// TIA Portal V20 export
FUNCTION_BLOCK "FB_LoaderShuttle2"   // FB205, SCL
{ S7_Optimized_Access := 'TRUE' }
// stored: AutoNumber false, MemoryReserve 100, SetENOAutomatically false
   VAR_INPUT
      iGripperReserved : Bool;
      iGripperReleased : Bool;
      iShuttleMoving : Bool;
      iShuttleInPos : Bool;
      iAxisV_Moving : Bool;
      iAxisV_InPos : Bool;
      iAxisW_Moving : Bool;
      iAxisW_InPos : Bool;
   END_VAR
   VAR_OUTPUT
      oExtGateOpenReq : Bool;
      oExtGateCloseReq : Bool;
      oIntGateOpenReq : Bool;
      oIntGateCloseReq : Bool;
      oLoadGripperCloseReq : Bool;
      oUnloadGripperOpenReq : Bool;
      oBlowingReq : Bool;
      oShuttleStartReq : Bool;
      oShuttlePosSetPoint : Real;
      oAxisVStartReq : Bool;
      oAxisVPosSetPoint : Real;
      oAxisWStartReq : Bool;
      oAxisWPosSetPoint : Real;
   END_VAR
   VAR
      sMain : "FB_Main";
      sShuttleInt { S7_SetPoint := 'True'} : "FB_ShuttleInt";
      sShuttleExt { S7_SetPoint := 'True'} : "FB_ShuttleExt";
      sControlIn { S7_SetPoint := 'True'} : "FB_PartControl";
      sControlOut { S7_SetPoint := 'True'} : "FB_PartControl";
      sBlowing { S7_SetPoint := 'True'} : "FB_Blowing";
      sIntLoadUnload { S7_SetPoint := 'True'} : "FB_IntLoadUnload";
      sExtLoadUnload { S7_SetPoint := 'True'} : "FB_ExtLoadUnload";
      sBwLoadUnload { S7_SetPoint := 'True'} : "FB_BwLoadUnload";
      sBwControlIn { S7_SetPoint := 'True'} : "FB_BwControl";
      sActPartControlIn { S7_SetPoint := 'True'} : "FB_ActControl";
      sActPartControlout { S7_SetPoint := 'True'} : "FB_ActControl";
      sActBwControlIn { S7_SetPoint := 'True'} : "FB_ActControl";
      sIntLoadUnloadOP { S7_SetPoint := 'True'} : "FB_IntLoadUnloadOP";
      sBwConsecutiveCtrl_1 { S7_SetPoint := 'True'} : "FB_Consecutive";
      sBwConsecutiveCtrl { S7_SetPoint := 'True'} : "FB_Consecutive";
      sShuttlePosInt { S7_SetPoint := 'True'} : Bool;
      sShuttlePosSas : Bool;
      sShuttlePosExt : Bool;
      sGripper_OK : Bool;
      sExtLoaderInSafePos : Bool;
      sIntLoaderInSafePos : Bool;
      sBwLoaderInSafePos : Bool;
      sRT_PartControlInMissing : R_TRIG;
      sRT_PartControlInExtra : R_TRIG;
      sRT_PartControlOutMissing : R_TRIG;
      sRT_PartControlOutExtra : R_TRIG;
      sRT_BwControlInMissing : R_TRIG;
      sRT_BwControlInExtra : R_TRIG;
      sStepPauseSeq { S7_SetPoint := 'True'} : Bool;
   END_VAR
   VAR_TEMP
      tAxis_U_Position : Struct
         ExtLoadUnloadAuto : Bool;
         ExtLoadUnloadManu : Bool;
         PartControl : Bool;
         BwLoad : Bool;
         BwUnload : Bool;
         BwControl : Bool;
         IntLoadUnload : Bool;
         Blowing : Bool;
         IntLoadUnloadOP : Bool;
      END_STRUCT;
      tAxis_V_Position : Struct
         LoadUnload : Bool;
         Safe : Bool;
         Blowing : Bool;
      END_STRUCT;
      tAxis_W_Position : Struct
         LoadUnload : Bool;
         Safe : Bool;
         Approach : Bool;
         Blowing : Bool;
      END_STRUCT;
   END_VAR
BEGIN
   REGION Shuttle 2 position
       // Init Position
       #sShuttlePosInt := FALSE;
       #sShuttlePosSas := FALSE;
       #sShuttlePosExt := FALSE;

       // Check Shuttle (U2 Axis) position
       IF "DB_AxisPosition".sAxis06_U2."$AA_IM" < "DB_AxisPosMachinePLC".Axis_U2.IntGateExt THEN
           #sShuttlePosExt := TRUE;
       ELSIF "DB_AxisPosition".sAxis06_U2."$AA_IM" > "DB_AxisPosMachinePLC".Axis_U2.ExtGateInt THEN
           #sShuttlePosInt := TRUE;
       ELSE
           #sShuttlePosSas := TRUE;
       END_IF;
   END_REGION

   REGION Position Check
       REGION Axis U2
           // Position : External Load / Unload Auto
           "FC_PositionCheck"(iAxisCurrentPos := "DB_AxisPosition".sAxis06_U2."$AA_IM",
                              iAxisTargetPos := "DB_AxisPosMachinePLC".Axis_U2.ExtLoadUnloadAuto,
                              iTolMin := 0.001,
                              iTolMax := 0.001,
                              iInPos => #tAxis_U_Position.ExtLoadUnloadAuto);

           // Position : External Load / Unload Manu
           "FC_PositionCheck"(iAxisCurrentPos := "DB_AxisPosition".sAxis06_U2."$AA_IM",
                              iAxisTargetPos := "DB_AxisPosMachinePLC".Axis_U2.ExtLoadUnloadManu,
                              iTolMin := 0.001,
                              iTolMax := 0.001,
                              iInPos => #tAxis_U_Position.ExtLoadUnloadManu);

           // Position : Part Control
           "FC_PositionCheck"(iAxisCurrentPos := "DB_AxisPosition".sAxis06_U2."$AA_IM",
                              iAxisTargetPos := "DB_AxisPosMachinePLC".Axis_U2.PartControl,
                              iTolMin := 0.001,
                              iTolMax := 0.001,
                              iInPos => #tAxis_U_Position.PartControl);

           // Position : Backwall Load
           "FC_PositionCheck"(iAxisCurrentPos := "DB_AxisPosition".sAxis06_U2."$AA_IM",
                              iAxisTargetPos := "DB_AxisPosMachinePLC".Axis_U2.BwLoad,
                              iTolMin := 0.001,
                              iTolMax := 0.001,
                              iInPos => #tAxis_U_Position.BwLoad);

           // Position : Backwall Unload
           "FC_PositionCheck"(iAxisCurrentPos := "DB_AxisPosition".sAxis06_U2."$AA_IM",
                              iAxisTargetPos := "DB_AxisPosMachinePLC".Axis_U2.BwUnLoad,
                              iTolMin := 0.001,
                              iTolMax := 0.001,
                              iInPos => #tAxis_U_Position.BwUnload);

           // Position : Backwall Control
           "FC_PositionCheck"(iAxisCurrentPos := "DB_AxisPosition".sAxis06_U2."$AA_IM",
                              iAxisTargetPos := "DB_AxisPosMachinePLC".Axis_U2.BwControl,
                              iTolMin := 0.001,
                              iTolMax := 0.001,
                              iInPos => #tAxis_U_Position.BwControl);

           // Position : Internal Load / Unload
           "FC_PositionCheck"(iAxisCurrentPos := "DB_AxisPosition".sAxis06_U2."$AA_IM",
                              iAxisTargetPos := "DB_AxisPosMachinePLC".Axis_U2.IntLoadUnload,
                              iTolMin := 0.001,
                              iTolMax := 0.001,
                              iInPos => #tAxis_U_Position.IntLoadUnload);

           // Position : Internal Load / Unload OP
           "FC_PositionCheck"(iAxisCurrentPos := "DB_AxisPosition".sAxis06_U2."$AA_IM",
                              iAxisTargetPos := "DB_AxisPosMachinePLC".Axis_U2.IntLoadUnloadOP,
                              iTolMin := 0.001,
                              iTolMax := 0.001,
                              iInPos => #tAxis_U_Position.IntLoadUnloadOP);

           // Position : Blowing (Undrilled part)
           "FC_PositionCheck"(iAxisCurrentPos := "DB_AxisPosition".sAxis06_U2."$AA_IM",
                              iAxisTargetPos := "DB_AxisPosMachinePLC".Axis_U2.Blowing,
                              iTolMin := 0.001,
                              iTolMax := 0.001,
                              iInPos => #tAxis_U_Position.Blowing);
       END_REGION

       REGION Axis V
           // Position : Load / Unload Auto
           "FC_PositionCheck"(iAxisCurrentPos := "DB_AxisPosition".sAxis07_V."$AA_IM",
                              iAxisTargetPos := "DB_AxisPosMachinePLC".Axis_V.Shuttle_2.LoadUnload,
                              iTolMin := 0.001,
                              iTolMax := 0.001,
                              iInPos => #tAxis_V_Position.LoadUnload);

           // Position : Safe
           "FC_PositionCheck"(iAxisCurrentPos := "DB_AxisPosition".sAxis07_V."$AA_IM",
                              iAxisTargetPos := "DB_AxisPosMachinePLC".Axis_V.Safe,
                              iTolMin := 0.001,
                              iTolMax := 0.001,
                              iInPos => #tAxis_V_Position.Safe);

           // Position : Blowing
           "FC_PositionCheck"(iAxisCurrentPos := "DB_AxisPosition".sAxis07_V."$AA_IM",
                              iAxisTargetPos := "DB_AxisPosMachinePLC".Axis_V.Shuttle_2.Blowing,
                              iTolMin := 0.001,
                              iTolMax := 0.001,
                              iInPos => #tAxis_V_Position.Blowing);
       END_REGION

       REGION Axis W
           // Position : Load / Unload Auto
           "FC_PositionCheck"(iAxisCurrentPos := "DB_AxisPosition".sAxis08_W."$AA_IM",
                              iAxisTargetPos := "DB_AxisPosMachinePLC".Axis_W.Shuttle_2.LoadUnload,
                              iTolMin := 0.001,
                              iTolMax := 0.001,
                              iInPos => #tAxis_W_Position.LoadUnload);

           // Position : Safe
           "FC_PositionCheck"(iAxisCurrentPos := "DB_AxisPosition".sAxis08_W."$AA_IM",
                              iAxisTargetPos := "DB_AxisPosMachinePLC".Axis_W.Safe,
                              iTolMin := 0.001,
                              iTolMax := 0.001,
                              iInPos => #tAxis_W_Position.Safe);

           // Position : Approach (confondu avec load/unload)
           "FC_PositionCheck"(iAxisCurrentPos := "DB_AxisPosition".sAxis08_W."$AA_IM",
                              iAxisTargetPos := "DB_AxisPosMachinePLC".Axis_W.Shuttle_2.Approach,
                              iTolMin := 0.001,
                              iTolMax := 0.001,
                              iInPos => #tAxis_W_Position.Approach);

           // Position : Blowing
           "FC_PositionCheck"(iAxisCurrentPos := "DB_AxisPosition".sAxis08_W."$AA_IM",
                              iAxisTargetPos := "DB_AxisPosMachinePLC".Axis_W.Shuttle_2.Blowing,
                              iTolMin := 0.001,
                              iTolMax := 0.001,
                              iInPos => #tAxis_W_Position.Blowing);
       END_REGION
   END_REGION

   REGION Step Pause Sequence
       #sStepPauseSeq := "LBP_ModeGroup".E_JOG
       OR "DB_CycleStartStop".sResquestStopNextCycle
       OR "LBP_Chan1".E_M01;

       #sMain.iStepPause := #sStepPauseSeq;
       #sShuttleInt.iStepPause := #sStepPauseSeq;
       #sShuttleExt.iStepPause := #sStepPauseSeq;
       #sIntLoadUnload.iStepPause := #sStepPauseSeq;
       #sIntLoadUnloadOP.iStepPause := #sStepPauseSeq;
       #sControlIn.iStepPause := #sStepPauseSeq;
       #sControlOut.iStepPause := #sStepPauseSeq;
       #sBwLoadUnload.iStepPause := #sStepPauseSeq;
       #sBwControlIn.iStepPause := #sStepPauseSeq;
       #sBlowing.iStepPause := #sStepPauseSeq;
       #sActPartControlIn.iStepPause := FALSE;
       #sActPartControlout.iStepPause := FALSE;
       #sActBwControlIn.iStepPause := FALSE;
   END_REGION

   REGION Main
       // Gripper prêt à Charger / Décharger une pièce
       #sGripper_OK :=
       ((("DB_PartManagement".sPosition.sShuttle2.Undrilled.Presence.Part AND NOT "DB_PartManagement".sPosition.sGripper.Undrilled.Presence.Part AND "DB_GestionGripper".sUndrilledGripper.oStateOpen) OR NOT "DB_PartManagement".sPosition.sShuttle2.Undrilled.Presence.Part)
       AND (("DB_PartManagement".sPosition.sGripper.Drilled.Presence.Part AND NOT "DB_PartManagement".sPosition.sShuttle2.Drilled.Presence.Part) OR NOT "DB_PartManagement".sPosition.sGripper.Drilled.Presence.Part));

       // Loader INT in Safe Position
       #sIntLoaderInSafePos := "DB_AxisPosition".sAxis07_V."$AA_IM" >= "DB_AxisPosMachinePLC".Axis_V.Safe
       OR ("DB_AxisPosition".sAxis07_V."$AA_IM" < "DB_AxisPosMachinePLC".Axis_V.Safe AND "DB_AxisPosition".sAxis08_W."$AA_IM" >= "DB_AxisPosMachinePLC".Axis_W.Safe);

       // Loader EXT in Safe Position
       #sExtLoaderInSafePos := "DB_SonplasMain".sSonplasLoader.iOperateInOutCollision;

       // BW Loader in Safe Position
       #sBwLoaderInSafePos := "DB_BwLoaderExchange".Inputs.BwLoaderInSafePos;

       // Test Stop after Emptying with only one Shuttle
       IF ("DB_WorkingModes".sEmptying
           AND NOT "DB_LoaderShuttle1".sMain.iJobReq
           AND "DB_PartManagement".sPosition.sPartNumber.Total <= 1) THEN
           #sMain.iJobReq := FALSE;
       END_IF;
       // Test Stop after Emptying with two Shuttle
       IF ("DB_WorkingModes".sEmptying
           AND "DB_LoaderShuttle1".sMain.iJobReq
           AND #sMain.sCurrent_Step_NB = 122
           AND "DB_PartManagement".sPosition.sPartNumber.Total <= 2) THEN
           #sMain.iJobReq := FALSE;
       END_IF;

       #sMain(iStartSeqCond := "DB_PowerOn".sMachineReadySoft AND NOT "MCP1_In".reset,
              iJobReq := #sMain.iJobReq,      
              iShuttleINT := #sShuttlePosInt,
              iShuttleSAS:= #sShuttlePosSas,
              iShuttleEXT := #sShuttlePosExt,
              iGripperReserved := #iGripperReserved,
              iGripperReleased := #iGripperReleased,
              iShuttleUndrilledPart:= "DB_PartManagement".sPosition.sShuttle2.Undrilled.Presence.Part,
              iShuttleDrilledPart:= "DB_PartManagement".sPosition.sShuttle2.Drilled.Presence.Part,
              iShuttleUndrilledBw:= "DB_PartManagement".sPosition.sShuttle2.Undrilled.Presence.BW,
              iShuttleDrilledBw:= "DB_PartManagement".sPosition.sShuttle2.Drilled.Presence.BW,
              iPartCtrlInOK:=#sControlIn.oPartControlOK,
              iPartCtrlInNOK:=#sControlIn.oPartControlNOK,
              iPartCtrlInContinuationStep:=#sActPartControlIn.oContinuationStep,
              iPartCtrlInRestartStep:=#sActPartControlIn.oRestartStep,
              iPartCtrlOutOK:=#sControlOut.oPartControlOK,
              iPartCtrlOutNOK:=#sControlOut.oPartControlNOK,
              iPartCtrlOutContinuationStep:=#sActPartControlout.oContinuationStep,
              iPartCtrlOutRestartStep:=#sActPartControlout.oRestartStep,
              iBwCtrlInOK:=#sBwControlIn.oBwControlOK,
              iBwCtrlInNOK:=#sBwControlIn.oBwControlNOK,
              iBwCtrlInContinuationStep:=#sActBwControlIn.oContinuationStep,
              iBwCtrlInRestartStep:=#sActBwControlIn.oRestartStep,
              iGripperOK:=#sGripper_OK,
              iNC_NoNeedAxis:=NOT "DB_CommPLC_ISO".sAxisManagedByNC,
              iExtLoaderInSafePos:=#sExtLoaderInSafePos,
              iIntLoaderInSafePos:=#sIntLoaderInSafePos,
              iBwLoaderInSafePos:=#sBwLoaderInSafePos,
              iOnePieceMode:="DB_WorkingModes".sOnePiece,
              iPLC_DateAndTime := "DB_ReadDateAndTime".sDateAndTime,
              iStepPause:=#sMain.iStepPause,
              oGripperAxisRequest => #sMain.oGripperAxisRequest,
              oGripperAxisRelease => #sMain.oGripperAxisRelease,
              oNoExtLoad=>#sMain.oNoExtLoad,
              oBwLoadReq=> #sMain.oBwLoadReq,
              oBwUnloadReq=> #sMain.oBwUnloadReq,
              ioShuttleIntSeq := #sShuttleInt.sInterface,
              ioShuttleExtSeq := #sShuttleExt.sInterface,
              ioControlInSeq := #sControlIn.sInterface,
              ioControlOutSeq := #sControlOut.sInterface,
              ioBlowingSeq:=#sBlowing.sInterface,
              ioIntLoadUnloadSeq := #sIntLoadUnload.sInterface,
              ioIntLoadUnloadOP_Seq:=#sIntLoadUnloadOP.sInterface,
              ioExtLoadUnloadSeq := #sExtLoadUnload.sInterface,
              ioBWLoadUnloadSeq := #sBwLoadUnload.sInterface,
              ioBWControlSeq := #sBwControlIn.sInterface,
              ioActPartControlInSeq:= #sActPartControlIn.sInterface,
              ioActPartControlOutSeq:= #sActPartControlout.sInterface,
              ioActBwControlInSeq:= #sActBwControlIn.sInterface);
   END_REGION

   REGION Msg Sequence Fault
       // Msg 700015 Shuttle 2 Sequence Fault
       IF #sMain.sCurrent_Step_NB = 999 THEN
           "LBP_AlarmMsgs".UserA[00].A70UUxx[15] := TRUE;
       END_IF;
   END_REGION

   REGION Shuttle 2 INT
       // Position INT :
       //  If Blowing : Pos. Blowing else Pos. Load/Unload
       IF "DB_LoaderOptions".Blowing.Disabled THEN
           #sShuttleInt.iShuttlePosIntSetPoint := "DB_AxisPosMachinePLC".Axis_U2.IntLoadUnload;
       ELSE
           #sShuttleInt.iShuttlePosIntSetPoint := "DB_AxisPosMachinePLC".Axis_U2.Blowing;
       END_IF;

       #sShuttleInt(iStartSeqCond := (#sMain.iStartSeqCond AND NOT #sShuttleInt.sInterface.Error AND NOT "DB_LoaderShuttle1".sShuttleInt.sInterface.SequenceRun AND #sShuttleInt.sInterface.StartRequest),
                    iJobReq := #sShuttleInt.sInterface.StartRequest,
                    iIntGateOpened := "DB_DigitalInputs".sInternalGateOpened.sSWStatus,
                    iIntGateClosed := "DB_DigitalInputs".sInternalGateLocked.sSWStatus,
                    iExtGateOpened := "DB_DigitalInputs".sExternalGateOpened.sSWStatus,
                    iExtGateClosed := "DB_DigitalInputs".sExternalGateLocked.sSWStatus,
                    iShuttlePosInt := #sShuttlePosInt,
                    iShuttlePosSas := #sShuttlePosSas,
                    iShuttlePosExt := #sShuttlePosExt,
                    iShuttlePosIntSetPoint := #sShuttleInt.iShuttlePosIntSetPoint,
                    iShuttlePosSasSetPoint := "DB_AxisPosMachinePLC".Axis_U2.Sas,
                    iShuttleMoving := #iShuttleMoving,
                    iShuttleInPos := #iShuttleInPos,
                    iIntLoaderInSafePos := #sIntLoaderInSafePos,
                    iPLC_DateAndTime:= "DB_ReadDateAndTime".sDateAndTime,
                    iStepPause:=#sShuttleInt.iStepPause,      
                    oExtGateOpenReq => #sShuttleInt.oExtGateOpenReq,
                    oExtGateCloseReq => #sShuttleInt.oExtGateCloseReq,
                    oIntGateOpenReq => #sShuttleInt.oIntGateOpenReq,
                    oIntGateCloseReq => #sShuttleInt.oIntGateCloseReq,
                    oShuttleStartReq => #sShuttleInt.oShuttleStartReq,
                    oShuttlePosSetPoint => #sShuttleInt.oShuttlePosSetPoint);
   END_REGION

   REGION Shuttle 2 EXT
       #sShuttleExt(iStartSeqCond := (#sIntLoaderInSafePos AND #sBwLoaderInSafePos AND #sMain.iStartSeqCond AND NOT #sShuttleExt.sInterface.Error AND NOT "DB_LoaderShuttle1".sShuttleExt.sInterface.SequenceRun AND #sShuttleExt.sInterface.StartRequest),
                    iJobReq := #sShuttleExt.sInterface.StartRequest,
                    iIntGateOpened := "DB_DigitalInputs".sInternalGateOpened.sSWStatus,
                    iIntGateClosed := "DB_DigitalInputs".sInternalGateLocked.sSWStatus,
                    iExtGateOpened := "DB_DigitalInputs".sExternalGateOpened.sSWStatus,
                    iExtGateClosed := "DB_DigitalInputs".sExternalGateLocked.sSWStatus,
                    iShuttlePosInt := #sShuttlePosInt,
                    iShuttlePosSas := #sShuttlePosSas,
                    iShuttlePosExt := #sShuttlePosExt,
                    iShuttlePosExtSetPoint := "DB_AxisPosMachinePLC".Axis_U2.BwUnLoad,
                    iShuttlePosSasSetPoint := "DB_AxisPosMachinePLC".Axis_U2.Sas,
                    iShuttleMoving := #iShuttleMoving,
                    iShuttleInPos := #iShuttleInPos,
                    iExtLoaderInSafePos := #sExtLoaderInSafePos,
                    iPLC_DateAndTime := "DB_ReadDateAndTime".sDateAndTime,
                    iStepPause:=#sShuttleExt.iStepPause,      
                    oExtGateOpenReq => #sShuttleExt.oExtGateOpenReq,
                    oExtGateCloseReq => #sShuttleExt.oExtGateCloseReq,
                    oIntGateOpenReq => #sShuttleExt.oIntGateOpenReq,
                    oIntGateCloseReq => #sShuttleExt.oIntGateCloseReq,
                    oShuttleStartReq => #sShuttleExt.oShuttleStartReq,
                    oShuttlePosSetPoint => #sShuttleExt.oShuttlePosSetPoint);
   END_REGION

   REGION Ext_LoadUnload
       #sExtLoadUnload(iStartSeqCond := (#sExtLoaderInSafePos AND #sMain.iStartSeqCond AND NOT #sExtLoadUnload.sInterface.Error AND NOT "DB_LoaderShuttle1".sExtLoadUnload.sInterface.SequenceRun AND #sExtLoadUnload.sInterface.StartRequest AND #sShuttlePosExt),
                       iJobReq := #sExtLoadUnload.sInterface.StartRequest,
                       iShuttleExtLoadUnloadAutoPos := #tAxis_U_Position.ExtLoadUnloadAuto,
                       iShuttleExtLoadUnloadAutoPosSetPoint := "DB_AxisPosMachinePLC".Axis_U2.ExtLoadUnloadAuto,
                       iShuttleExtLoadUnloadManuPos := #tAxis_U_Position.ExtLoadUnloadManu,
                       iShuttleExtLoadUnloadManuPosSetPoint := "DB_AxisPosMachinePLC".Axis_U2.ExtLoadUnloadManu,
                       iShuttleMoving := #iShuttleMoving,
                       iShuttleInPos := #iShuttleInPos,
                       iCommunicationWithExtLoaderDone := "DB_SonplasMain".sSonplasLoader.iPartInShuttle2Finished,
                       iLoadUnloadMsgManuModeAck := #sExtLoadUnload.iLoadUnloadMsgManuModeAck OR "MCP1_In".plus OR "DI_SemiAutoValid", // WFA TBD
                       iAutoMode := "DB_WorkingModes".sAuto,
                       iSemiAutoMode := "DB_WorkingModes".sSemiAuto,
                       iFillingMode := "DB_WorkingModes".sFilling AND NOT #sMain.oNoExtLoad,
                       iEmptyingMode := "DB_WorkingModes".sEmptying OR #sMain.oNoExtLoad,
                       iPLC_DateAndTime:= "DB_ReadDateAndTime".sDateAndTime,
                       iStepPause:=#sExtLoadUnload.iStepPause,      
                       oShuttleStartReq => #sExtLoadUnload.oShuttleStartReq,
                       oShuttlePosSetPoint => #sExtLoadUnload.oShuttlePosSetPoint,
                       oStartCommunicationWithExtLoader => "DB_SonplasMain".sSonplasLoader.oPartOutShuttle2InPos,
                       oSetLoadUnloadMsgManuMode => #sExtLoadUnload.oSetLoadUnloadMsgManuMode);

       // Message "Part loaded by operator"
       // IF #sExtLoadUnload.oSetLoadUnloadMsgManuMode THEN
       //     "LBP_AlarmMsgs".UserA[00].A70UUxx[55] := TRUE;
       // ELSIF
       //     #sExtLoadUnload.iLoadUnloadMsgManuModeAck OR "LBP_Chan1".A_Reset THEN
       //     "LBP_AlarmMsgs".UserA[00].A70UUxx[55] := FALSE;
       // END_IF;
       "LBP_AlarmMsgs".UserA[00].A70UUxx[55] := FALSE;
        #sExtLoadUnload.iLoadUnloadMsgManuModeAck := FALSE;
   END_REGION

   REGION Int_LoadUnload
       // Load Gripper Closed according to dry run working mode
        #sIntLoadUnload.iLoadGripperClosed := ("DB_GestionGripper".sUndrilledGripper.oStateCloseWithPart AND NOT "DB_WorkingModes".sDryRun) 
       OR ("DB_GestionGripper".sUndrilledGripper.oStateClose AND "DB_WorkingModes".sDryRun);

       #sIntLoadUnload(iStartSeqCond := (#sIntLoaderInSafePos AND #sMain.iStartSeqCond AND NOT #sIntLoadUnload.sInterface.Error AND NOT "DB_LoaderShuttle1".sIntLoadUnload.sInterface.SequenceRun AND #sIntLoadUnload.sInterface.StartRequest AND #sShuttlePosInt),
                       iJobReq := #sIntLoadUnload.sInterface.StartRequest,
                       iShuttleIntLoadUnloadPos := #tAxis_U_Position.IntLoadUnload,
                       iShuttleIntLoadUnloadPosSetPoint := "DB_AxisPosMachinePLC".Axis_U2.IntLoadUnload,
                       iAxisV_LoadUnloadShuttlePos := #tAxis_V_Position.LoadUnload,
                       iAxisV_LoadUnloadShuttlePosSetPoint := "DB_AxisPosMachinePLC".Axis_V.Shuttle_2.LoadUnload,
                       iAxisV_SafePos := #tAxis_V_Position.Safe,
                       iAxisV_SafePosSetPoint := "DB_AxisPosMachinePLC".Axis_V.Safe,
                       iAxisW_SafePos := #tAxis_W_Position.Safe,
                       iAxisW_SafePosSetPoint := "DB_AxisPosMachinePLC".Axis_W.Safe,
                       iAxisW_ApproachLoadUnloadPos := #tAxis_W_Position.Approach,
                       iAxisW_ApproachLoadUnloadSetPoint := "DB_AxisPosMachinePLC".Axis_W.Shuttle_2.Approach,
                       iAxisW_LoadUnloadPos := #tAxis_W_Position.LoadUnload,
                       iAxisW_LoadUnloadPosSetPoint := "DB_AxisPosMachinePLC".Axis_W.Shuttle_2.LoadUnload,
                       iShuttleMoving := #iShuttleMoving,
                       iShuttleInPos := #iShuttleInPos,
                       iAxisV_Moving := #iAxisV_Moving,
                       iAxisW_InPos := #iAxisW_InPos,
                       iAxisV_InPos := #iAxisV_InPos,
                       iAxisW_Moving := #iAxisW_Moving,
                       iDrilledPartToUnload:= "DB_PartManagement".sPosition.sGripper.Drilled.Presence.Part,
                       iUnDrilledPartToLoad:= "DB_PartManagement".sPosition.sShuttle2.Undrilled.Presence.Part,
                       iLoadGripperClosed := #sIntLoadUnload.iLoadGripperClosed,
                       iUnloadGripperOpen := "DB_GestionGripper".sDrilledGripper.oStateOpen,
                       iPLC_DateAndTime:= "DB_ReadDateAndTime".sDateAndTime,
                       iStepPause:=#sIntLoadUnload.iStepPause,      
                       oShuttleStartReq => #sIntLoadUnload.oShuttleStartReq,
                       oShuttlePosSetPoint => #sIntLoadUnload.oShuttlePosSetPoint,
                       oAxisV_StartReq => #sIntLoadUnload.oAxisV_StartReq,
                       oAxisV_PosSetPoint => #sIntLoadUnload.oAxisV_PosSetPoint,
                       oAxisW_StartReq => #sIntLoadUnload.oAxisW_StartReq,
                       oAxisW_PosSetPoint => #sIntLoadUnload.oAxisW_PosSetPoint,
                       oLoadGripperCloseReq => #sIntLoadUnload.oLoadGripperCloseReq,
                       oUnloadGripperOpenReq => #sIntLoadUnload.oUnloadGripperOpenReq);
   END_REGION

   REGION Int_LoadUnloadOP
           // Load Gripper Closed according to dry run working mode
            #sIntLoadUnloadOP.iLoadGripperClosed := ("DB_GestionGripper".sUndrilledGripper.oStateCloseWithPart AND NOT "DB_WorkingModes".sDryRun) // WFA A Remettre
            OR ("DB_GestionGripper".sUndrilledGripper.oStateClose AND "DB_WorkingModes".sDryRun);

    #sIntLoadUnloadOP(iStartSeqCond := (#sIntLoaderInSafePos AND #sMain.iStartSeqCond AND NOT #sIntLoadUnloadOP.sInterface.Error AND NOT "DB_LoaderShuttle1".sIntLoadUnloadOP.sInterface.SequenceRun AND #sIntLoadUnloadOP.sInterface.StartRequest AND #sShuttlePosInt),
                      iJobReq := #sIntLoadUnloadOP.sInterface.StartRequest,
                      iShuttleIntLoadUnloadPos := #tAxis_U_Position.IntLoadUnload,
                      iShuttleIntLoadUnloadPosSetPoint := "DB_AxisPosMachinePLC".Axis_U2.IntLoadUnload,
                      iShuttleIntLoadUnloadOP_Pos:=#tAxis_U_Position.IntLoadUnloadOP,
                      iShuttleIntLoadUnloadOP_PosSetPoint:="DB_AxisPosMachinePLC".Axis_U2.IntLoadUnloadOP,
                      iAxisV_LoadUnloadShuttlePos := #tAxis_V_Position.LoadUnload,
                      iAxisV_LoadUnloadShuttlePosSetPoint := "DB_AxisPosMachinePLC".Axis_V.Shuttle_2.LoadUnload,
                      iAxisV_SafePos := #tAxis_V_Position.Safe,
                      iAxisV_SafePosSetPoint := "DB_AxisPosMachinePLC".Axis_V.Safe,
                      iAxisW_SafePos := #tAxis_W_Position.Safe,
                      iAxisW_SafePosSetPoint := "DB_AxisPosMachinePLC".Axis_W.Safe,
                      iAxisW_ApproachLoadUnloadPos := #tAxis_W_Position.Approach,
                      iAxisW_ApproachLoadUnloadSetPoint := "DB_AxisPosMachinePLC".Axis_W.Shuttle_2.Approach,
                      iAxisW_LoadUnloadPos := #tAxis_W_Position.LoadUnload,
                      iAxisW_LoadUnloadPosSetPoint := "DB_AxisPosMachinePLC".Axis_W.Shuttle_2.LoadUnload,
                      iShuttleMoving := #iShuttleMoving,
                      iShuttleInPos := #iShuttleInPos,
                      iAxisV_Moving := #iAxisV_Moving,
                      iAxisW_InPos := #iAxisW_InPos,
                      iAxisV_InPos := #iAxisV_InPos,
                      iAxisW_Moving := #iAxisW_Moving,
                      iDrilledPartToUnload := "DB_PartManagement".sPosition.sGripper.Drilled.Presence.Part,
                      iUnDrilledPartToLoad := "DB_PartManagement".sPosition.sShuttle2.Undrilled.Presence.Part,
                      iLoadGripperClosed := #sIntLoadUnloadOP.iLoadGripperClosed,
                      iUnloadGripperOpen := "DB_GestionGripper".sDrilledGripper.oStateOpen,
                      iPLC_DateAndTime := "DB_ReadDateAndTime".sDateAndTime,
                      iStepPause := #sIntLoadUnloadOP.iStepPause,        
                      oShuttleStartReq => #sIntLoadUnloadOP.oShuttleStartReq,
                      oShuttlePosSetPoint => #sIntLoadUnloadOP.oShuttlePosSetPoint,
                      oAxisV_StartReq => #sIntLoadUnloadOP.oAxisV_StartReq,
                      oAxisV_PosSetPoint => #sIntLoadUnloadOP.oAxisV_PosSetPoint,
                      oAxisW_StartReq => #sIntLoadUnloadOP.oAxisW_StartReq,
                      oAxisW_PosSetPoint => #sIntLoadUnloadOP.oAxisW_PosSetPoint,
                      oLoadGripperCloseReq => #sIntLoadUnloadOP.oLoadGripperCloseReq,
                      oUnloadGripperOpenReq => #sIntLoadUnloadOP.oUnloadGripperOpenReq);
   END_REGION

   REGION Parts Control
       // Control In

       // Expected control result
       IF "DB_WorkingModes".sFilling THEN
           #sControlIn.iExpectedCtrlUndrilled := TRUE;
           #sControlIn.iExpectedCtrlDrilled := FALSE;
       ELSIF "DB_WorkingModes".sNormal THEN
           #sControlIn.iExpectedCtrlUndrilled := TRUE;
           #sControlIn.iExpectedCtrlDrilled := FALSE;
       ELSIF "DB_WorkingModes".sEmptying THEN
           #sControlIn.iExpectedCtrlUndrilled := FALSE;
           #sControlIn.iExpectedCtrlDrilled := FALSE;
       END_IF;

       #sControlIn(iStartSeqCond := (#sExtLoaderInSafePos AND #sMain.iStartSeqCond AND NOT #sControlIn.sInterface.Error AND NOT "DB_LoaderShuttle1".sControlIn.sInterface.SequenceRun AND #sControlIn.sInterface.StartRequest AND #sShuttlePosExt),
                   iJobReq := #sControlIn.sInterface.StartRequest,
                   iCtrlEnabled := TRUE,
                   iShuttleCtrlPos := #tAxis_U_Position.PartControl,
                   iShuttleCtrlPosSetPoint := "DB_AxisPosMachinePLC".Axis_U2.PartControl,
                   iExpectedCtrlUndrilled := #sControlIn.iExpectedCtrlUndrilled,
                   iExpectedCtrlDrilled := #sControlIn.iExpectedCtrlDrilled,
                   iUndrilledPartPresence:= "DB_DigitalInputsBW_Station".sUndrilledPartCtrl.sSWStatus,
                   iDrilledPartPresence:= "DB_DigitalInputsBW_Station".sDrilledPartCtrl.sSWStatus,
                   iShuttleMoving := #iShuttleMoving,
                   iShuttleInPos := #iShuttleInPos,
                   iPLC_DateAndTime := "DB_ReadDateAndTime".sDateAndTime,
                   iStepPause := #sControlIn.iStepPause,       
                   oShuttleStartReq => #sControlIn.oShuttleStartReq,
                   oShuttlePosSetPoint => #sControlIn.oShuttlePosSetPoint,
                   oPartControlOK => #sControlIn.oPartControlOK,
                   oPartControlNOK => #sControlIn.oPartControlNOK);

       // Control Out

       // Expected control result
       #sControlOut.iExpectedCtrlUndrilled := "DB_PartManagement".sPosition.sShuttle2.Undrilled.Presence.Part;
       #sControlOut.iExpectedCtrlDrilled := "DB_PartManagement".sPosition.sShuttle2.Drilled.Presence.Part;

       #sControlOut(iStartSeqCond := (#sBwLoaderInSafePos AND #sMain.iStartSeqCond AND NOT #sControlOut.sInterface.Error AND NOT "DB_LoaderShuttle1".sControlOut.sInterface.SequenceRun AND #sControlOut.sInterface.StartRequest AND #sShuttlePosExt),
                    iJobReq := #sControlOut.sInterface.StartRequest,
                    iCtrlEnabled := TRUE,
                    iShuttleCtrlPos := #tAxis_U_Position.PartControl,
                    iShuttleCtrlPosSetPoint := "DB_AxisPosMachinePLC".Axis_U2.PartControl,
                    iExpectedCtrlUndrilled := #sControlOut.iExpectedCtrlUndrilled,
                    iExpectedCtrlDrilled := #sControlOut.iExpectedCtrlDrilled,
                    iUndrilledPartPresence:="DB_DigitalInputsBW_Station".sUndrilledPartCtrl.sSWStatus,
                    iDrilledPartPresence:="DB_DigitalInputsBW_Station".sDrilledPartCtrl.sSWStatus,
                    iShuttleMoving := #iShuttleMoving,
                    iShuttleInPos := #iShuttleInPos,
                    iPLC_DateAndTime := "DB_ReadDateAndTime".sDateAndTime,
                    iStepPause := #sControlOut.iStepPause,      
                    oShuttleStartReq => #sControlOut.oShuttleStartReq,
                    oShuttlePosSetPoint => #sControlOut.oShuttlePosSetPoint,
                    oPartControlOK => #sControlOut.oPartControlOK,
                    oPartControlNOK => #sControlOut.oPartControlNOK);
   END_REGION

   REGION BW Load Unload
       #sBwLoadUnload(iStartSeqCond := (#sMain.iStartSeqCond AND NOT #sBwLoadUnload.sInterface.Error AND NOT "DB_LoaderShuttle1".sBwLoadUnload.sInterface.SequenceRun AND #sBwLoadUnload.sInterface.StartRequest AND #sShuttlePosExt),
                      iJobReq := #sBwLoadUnload.sInterface.StartRequest,
                      iLoadReq:= #sMain.oBwLoadReq,
                      iUnloadReq:= #sMain.oBwUnloadReq,
                      iShuttleBwUnloadPos := #tAxis_U_Position.BwUnload,
                      iShuttleBwUnloadPosSetPoint := "DB_AxisPosMachinePLC".Axis_U2.BwUnLoad,
                      iShuttleBwLoadPos := #tAxis_U_Position.BwLoad,
                      iShuttleBwLoadPosSetPoint := "DB_AxisPosMachinePLC".Axis_U2.BwLoad,
                      iShuttleMoving := #iShuttleMoving,
                      iShuttleInPos := #iShuttleInPos,
                      iBwLoadDone:= "DB_BwLoader".sBwCommunication.oLoadJobDone,
                      iBwUnloadDone:= "DB_BwLoader".sBwCommunication.oUnloadJobDone,
                      iBwLoaderInSafePos:=#sBwLoaderInSafePos,
                      iPLC_DateAndTime:= "DB_ReadDateAndTime".sDateAndTime,
                      iStepPause:=#sBwLoadUnload.iStepPause,      
                      oShuttleStartReq => #sBwLoadUnload.oShuttleStartReq,
                      oShuttlePosSetPoint => #sBwLoadUnload.oShuttlePosSetPoint,
                      oBwLoadReq=>#sBwLoadUnload.oBwLoadReq,
                      oBwUnloadReq=>#sBwLoadUnload.oBwUnloadReq);
   END_REGION

   REGION BW Control
       // BW Control In

       // Expected control result
       #sBwControlIn.iExpectedCtrl := "DB_PartManagement".sPosition.sShuttle2.Undrilled.Presence.Part;

       #sBwControlIn(iStartSeqCond := (#sMain.iStartSeqCond AND NOT #sBwControlIn.sInterface.Error AND NOT "DB_LoaderShuttle1".sBwControlIn.sInterface.SequenceRun AND #sBwControlIn.sInterface.StartRequest AND #sShuttlePosExt),
                     iJobReq := #sBwControlIn.sInterface.StartRequest,
                     iCtrlEnabled := TRUE,
                     iShuttleCtrlPos := #tAxis_U_Position.BwControl,
                     iShuttleCtrlPosSetPoint := "DB_AxisPosMachinePLC".Axis_U2.BwControl,
                     iExpectedCtrl := #sBwControlIn.iExpectedCtrl,
                     iBwPresence := "DB_DigitalInputsBW_Station".sBwCtrl.sSWStatus,
                     iShuttleMoving := #iShuttleMoving,
                     iShuttleInPos := #iShuttleInPos,
                     iPLC_DateAndTime := "DB_ReadDateAndTime".sDateAndTime,
                     iStepPause := #sBwControlIn.iStepPause,   
                     oShuttleStartReq => #sBwControlIn.oShuttleStartReq,
                     oShuttlePosSetPoint => #sBwControlIn.oShuttlePosSetPoint,
                     oBwControlOK => #sBwControlIn.oBwControlOK,
                     oBwControlNOK => #sBwControlIn.oBwControlNOK);

       #sBwConsecutiveCtrl(iReset := #sBwConsecutiveCtrl.oConsecutiveError AND #sActBwControlIn.sCurrent_Step_NB = 60,
                           iGoodEntry := #sBwControlIn.oBwControlOK,
                           iBadEntry := #sBwControlIn.oBwControlNOK,
                           iPresetValue := 3,
                           oConsecutiveError => #sBwConsecutiveCtrl.oConsecutiveError);
   END_REGION

   REGION Blowing
       #sBlowing(iStartSeqCond := (#sIntLoaderInSafePos AND #sMain.iStartSeqCond AND NOT #sBlowing.sInterface.Error AND NOT "DB_LoaderShuttle1".sBlowing.sInterface.SequenceRun AND #sBlowing.sInterface.StartRequest AND #sShuttlePosInt),
                 iJobReq := #sBlowing.sInterface.StartRequest,
                 iShuttleBlowingPos := #tAxis_U_Position.Blowing,
                 iShuttleBlowingPosSetPoint := "DB_AxisPosMachinePLC".Axis_U2.Blowing,
                 iAxisV_BlowingPos := #tAxis_V_Position.Blowing,
                 iAxisV_BlowingPosSetPoint := "DB_AxisPosMachinePLC".Axis_V.Shuttle_2.Blowing,
                 iAxisW_SafePos := #tAxis_W_Position.Safe,
                 iAxisW_SafePosSetPoint := "DB_AxisPosMachinePLC".Axis_W.Safe,
                 iAxisW_BlowingPos := #tAxis_W_Position.Blowing,
                 iAxisW_BlowingPosSetPoint := "DB_AxisPosMachinePLC".Axis_W.Shuttle_2.Blowing,
                 iShuttleMoving := #iShuttleMoving,
                 iShuttleInPos := #iShuttleInPos,
                 iAxisV_Moving := #iAxisV_Moving,
                 iAxisV_InPos := #iAxisV_InPos,
                 iAxisW_Moving := #iAxisW_Moving,
                 iAxisW_InPos := #iAxisW_InPos,
                 iBlowingTime:=DINT_TO_TIME(REAL_TO_DINT("DB_HMISetting".BlowingSetpoint)),
                 iPLC_DateAndTime := "DB_ReadDateAndTime".sDateAndTime,
                 iStepPause := #sBlowing.iStepPause,
                 oShuttleStartReq => #sBlowing.oShuttleStartReq,
                 oShuttlePosSetPoint => #sBlowing.oShuttlePosSetPoint,
                 oAxisV_StartReq => #sBlowing.oAxisV_StartReq,
                 oAxisV_PosSetPoint => #sBlowing.iAxisV_BlowingPosSetPoint,
                 oAxisW_StartReq => #sBlowing.oAxisW_StartReq,
                 oAxisW_PosSetPoint => #sBlowing.iAxisW_BlowingPosSetPoint,
                 oBlowingReq => #sBlowing.oBlowingReq);
   END_REGION

   REGION Action Part Control In
       // Conditions d'arrêt en Mode Auto
       #sActPartControlIn.iModeAutoPosCondition :=
       ("DB_WorkingModes".sAuto AND (#sControlIn.sMissingPartCtrlUndrilled OR #sControlIn.sMissingPartCtrlDrilled) AND "DB_LoaderOptions".ActPartControlIn.Stop)
       OR ("DB_WorkingModes".sAuto AND (#sControlIn.sExtraPartCtrlUndrilled OR #sControlIn.sExtraPartCtrlDrilled) AND "DB_LoaderOptions".ActPartControlIn.Stop)
       OR ("DB_WorkingModes".sAuto AND (#sControlIn.sExtraPartCtrlUndrilled OR #sControlIn.sExtraPartCtrlDrilled) AND NOT "DB_LoaderOptions".ActPartControlIn.Stop);
       // Conditions d'arrêt en Mode Semi Auto   
       #sActPartControlIn.iModeSemiAutoPosCondition :=
       ("DB_WorkingModes".sSemiAuto AND (#sControlIn.sMissingPartCtrlUndrilled OR #sControlIn.sMissingPartCtrlDrilled) AND "DB_LoaderOptions".ActPartControlIn.Stop)
       OR ("DB_WorkingModes".sSemiAuto AND (#sControlIn.sExtraPartCtrlUndrilled OR #sControlIn.sExtraPartCtrlDrilled) AND "DB_LoaderOptions".ActPartControlIn.Stop)
       OR ("DB_WorkingModes".sSemiAuto AND (#sControlIn.sExtraPartCtrlUndrilled OR #sControlIn.sExtraPartCtrlDrilled) AND NOT "DB_LoaderOptions".ActPartControlIn.Stop);
       // Conditions pas d'arrêt
       #sActPartControlIn.iNoStopCondition :=
       ("DB_WorkingModes".sAuto AND (#sControlIn.sMissingPartCtrlUndrilled OR #sControlIn.sMissingPartCtrlDrilled) AND NOT "DB_LoaderOptions".ActPartControlIn.Stop)
       OR ("DB_WorkingModes".sSemiAuto AND (#sControlIn.sMissingPartCtrlUndrilled OR #sControlIn.sMissingPartCtrlDrilled) AND NOT "DB_LoaderOptions".ActPartControlIn.Stop);

       #sActPartControlIn(iStartSeqCond := (#sMain.iStartSeqCond AND NOT #sActPartControlIn.sInterface.Error AND NOT "DB_LoaderShuttle1".sActPartControlIn.sInterface.SequenceRun AND #sActPartControlIn.sInterface.StartRequest AND #sShuttlePosExt),
                          iJobReq := #sActPartControlIn.sInterface.StartRequest,
                          iShuttleModeAutoPos := #tAxis_U_Position.ExtLoadUnloadAuto,
                          iShuttleModeAutoPosSetPoint := "DB_AxisPosMachinePLC".Axis_U2.ExtLoadUnloadAuto,
                          iShuttleModeSemiAutoPos := #tAxis_U_Position.ExtLoadUnloadManu,
                          iShuttleModeSemiAutoPosSetPoint := "DB_AxisPosMachinePLC".Axis_U2.ExtLoadUnloadManu,
                          iShuttleMoving := #iShuttleMoving,
                          iShuttleInPos := #iShuttleInPos,
                          iModeAutoPosCondition := #sActPartControlIn.iModeAutoPosCondition,
                          iModeSemiAutoPosCondition := #sActPartControlIn.iModeSemiAutoPosCondition,
                          iNoStopCondition := #sActPartControlIn.iNoStopCondition,
                          iOperatorCycleRestart := "LBP_Chan1".E_ProgRunning,
                          iNC_Stopped := NOT "LBP_Chan1".E_ProgRunning,
                          iNC_Running := "LBP_Chan1".E_ProgRunning,
                          iMissingPart:=#sControlIn.sMissingPartCtrlUndrilled OR #sControlIn.sMissingPartCtrlDrilled,
                          iExtraPart:=#sControlIn.sExtraPartCtrlUndrilled OR #sControlIn.sExtraPartCtrlDrilled,
                          iPLC_DateAndTime := "DB_ReadDateAndTime".sDateAndTime,
                          iStepPause := #sActPartControlIn.iStepPause,
                          oShuttleStartReq => #sActPartControlIn.oShuttleStartReq,
                          oShuttlePosSetPoint => #sActPartControlIn.oShuttlePosSetPoint,
                          oStopNC_Req => #sActPartControlIn.oStopNC_Req,       // Implicite par Alarm Message
                          oRestartNC_Req => #sActPartControlIn.oRestartNC_Req, // Implicite par Restart NC
                          oRestartStep => #sActPartControlIn.oRestartStep,
                          oContinuationStep => #sActPartControlIn.oContinuationStep,
                          oMsgMissingPart=>#sActPartControlIn.oMsgMissingPart,
                          oMsgExtraPart=>#sActPartControlIn.oMsgExtraPart);

       #sRT_PartControlInMissing(CLK := #sActPartControlIn.oMsgMissingPart);
       IF #sRT_PartControlInMissing.Q THEN
           "LBP_AlarmMsgs".UserA[03].A70UUxx[21] := TRUE;
       END_IF;

       #sRT_PartControlInExtra(CLK := #sActPartControlIn.oMsgExtraPart);
       IF #sRT_PartControlInExtra.Q THEN
           "LBP_AlarmMsgs".UserA[03].A70UUxx[22] := TRUE;
       END_IF;
   END_REGION

   REGION Action Part Control Out
       // Conditions d'arrêt en Mode Auto
       #sActPartControlout.iModeAutoPosCondition :=
       ("DB_WorkingModes".sAuto AND (#sControlOut.sMissingPartCtrlUndrilled OR #sControlOut.sMissingPartCtrlDrilled) AND "DB_LoaderOptions".ActPartControlOut.Stop)
       OR ("DB_WorkingModes".sAuto AND (#sControlOut.sExtraPartCtrlUndrilled OR #sControlOut.sExtraPartCtrlDrilled) AND "DB_LoaderOptions".ActPartControlOut.Stop)
       OR ("DB_WorkingModes".sAuto AND (#sControlOut.sExtraPartCtrlUndrilled OR #sControlOut.sExtraPartCtrlDrilled) AND NOT "DB_LoaderOptions".ActPartControlOut.Stop);
       // Conditions d'arrêt en Mode Semi Auto 
       #sActPartControlout.iModeSemiAutoPosCondition :=
       ("DB_WorkingModes".sSemiAuto AND (#sControlOut.sMissingPartCtrlUndrilled OR #sControlOut.sMissingPartCtrlDrilled) AND "DB_LoaderOptions".ActPartControlOut.Stop)
       OR ("DB_WorkingModes".sSemiAuto AND (#sControlOut.sExtraPartCtrlUndrilled OR #sControlOut.sExtraPartCtrlDrilled) AND "DB_LoaderOptions".ActPartControlOut.Stop)
       OR ("DB_WorkingModes".sSemiAuto AND (#sControlOut.sExtraPartCtrlUndrilled OR #sControlOut.sExtraPartCtrlDrilled) AND NOT "DB_LoaderOptions".ActPartControlOut.Stop);
       // Conditions pas d'arrêt
       #sActPartControlout.iNoStopCondition :=
       ("DB_WorkingModes".sAuto AND (#sControlOut.sMissingPartCtrlUndrilled OR #sControlOut.sMissingPartCtrlDrilled) AND NOT "DB_LoaderOptions".ActPartControlOut.Stop)
       OR ("DB_WorkingModes".sSemiAuto AND (#sControlOut.sMissingPartCtrlUndrilled OR #sControlOut.sMissingPartCtrlDrilled) AND NOT "DB_LoaderOptions".ActPartControlOut.Stop);

       #sActPartControlout(iStartSeqCond := (#sMain.iStartSeqCond AND NOT #sActPartControlout.sInterface.Error AND NOT "DB_LoaderShuttle1".sActPartControlOut.sInterface.SequenceRun AND #sActPartControlout.sInterface.StartRequest AND #sShuttlePosExt),
                           iJobReq := #sActPartControlout.sInterface.StartRequest,
                           iShuttleModeAutoPos := #tAxis_U_Position.ExtLoadUnloadAuto,
                           iShuttleModeAutoPosSetPoint := "DB_AxisPosMachinePLC".Axis_U2.ExtLoadUnloadAuto,
                           iShuttleModeSemiAutoPos := #tAxis_U_Position.ExtLoadUnloadManu,
                           iShuttleModeSemiAutoPosSetPoint := "DB_AxisPosMachinePLC".Axis_U2.ExtLoadUnloadManu,
                           iShuttleMoving := #iShuttleMoving,
                           iShuttleInPos := #iShuttleInPos,
                           iModeAutoPosCondition := #sActPartControlout.iModeAutoPosCondition,
                           iModeSemiAutoPosCondition := #sActPartControlout.iModeSemiAutoPosCondition,
                           iNoStopCondition := #sActPartControlout.iNoStopCondition,
                           iOperatorCycleRestart := "LBP_Chan1".E_ProgRunning,
                           iNC_Stopped := NOT "LBP_Chan1".E_ProgRunning,
                           iNC_Running := "LBP_Chan1".E_ProgRunning,
                           iMissingPart:=#sControlOut.sMissingPartCtrlUndrilled OR #sControlOut.sMissingPartCtrlDrilled,
                           iExtraPart:=#sControlOut.sExtraPartCtrlUndrilled OR #sControlOut.sExtraPartCtrlDrilled,
                           iPLC_DateAndTime := "DB_ReadDateAndTime".sDateAndTime,
                           iStepPause := #sActPartControlout.iStepPause,
                           oShuttleStartReq => #sActPartControlout.oShuttleStartReq,
                           oShuttlePosSetPoint => #sActPartControlout.oShuttlePosSetPoint,
                           oStopNC_Req => #sActPartControlout.oStopNC_Req,       // Implicite par Alarm Message
                           oRestartNC_Req => #sActPartControlout.oRestartNC_Req, // Implicite par Restart NC
                           oRestartStep => #sActPartControlout.oRestartStep,
                           oContinuationStep => #sActPartControlout.oContinuationStep,
                           oMsgMissingPart=>#sActPartControlout.oMsgMissingPart,
                           oMsgExtraPart=>#sActPartControlout.oMsgExtraPart);

       #sRT_PartControlOutMissing(CLK := #sActPartControlout.oMsgMissingPart);
       IF #sRT_PartControlOutMissing.Q THEN
           "LBP_AlarmMsgs".UserA[03].A70UUxx[23] := TRUE;
       END_IF;

       #sRT_PartControlOutExtra(CLK := #sActPartControlout.oMsgExtraPart);
       IF #sRT_PartControlOutExtra.Q THEN
           "LBP_AlarmMsgs".UserA[03].A70UUxx[24] := TRUE;
       END_IF;
   END_REGION

   REGION Action Bw Control In
       // Conditions d'arrêt en Mode Auto
       #sActBwControlIn.iModeAutoPosCondition :=
       ("DB_WorkingModes".sAuto AND #sBwControlIn.sMissingBwCtrl AND ("DB_LoaderOptions".ActBwControlIn.Stop OR #sBwConsecutiveCtrl.oConsecutiveError))
       OR ("DB_WorkingModes".sAuto AND #sBwControlIn.sExtraBwCtrl AND "DB_LoaderOptions".ActBwControlIn.Stop)
       OR ("DB_WorkingModes".sAuto AND #sBwControlIn.sExtraBwCtrl AND NOT "DB_LoaderOptions".ActBwControlIn.Stop);
       // Conditions d'arrêt en Mode Semi Auto
       #sActBwControlIn.iModeSemiAutoPosCondition :=
       ("DB_WorkingModes".sSemiAuto AND #sBwControlIn.sMissingBwCtrl AND "DB_LoaderOptions".ActBwControlIn.Stop)
       OR ("DB_WorkingModes".sSemiAuto AND #sBwControlIn.sExtraBwCtrl AND "DB_LoaderOptions".ActBwControlIn.Stop)
       OR ("DB_WorkingModes".sSemiAuto AND #sBwControlIn.sExtraBwCtrl AND NOT "DB_LoaderOptions".ActBwControlIn.Stop);
       // Conditions pas d'arrêt
       #sActBwControlIn.iNoStopCondition :=
       ("DB_WorkingModes".sAuto AND #sBwControlIn.sMissingBwCtrl AND (NOT "DB_LoaderOptions".ActBwControlIn.Stop AND NOT #sBwConsecutiveCtrl.oConsecutiveError))
       OR ("DB_WorkingModes".sSemiAuto AND #sBwControlIn.sMissingBwCtrl AND NOT "DB_LoaderOptions".ActBwControlIn.Stop);

       #sActBwControlIn(iStartSeqCond := (#sMain.iStartSeqCond AND NOT #sActBwControlIn.sInterface.Error AND NOT "DB_LoaderShuttle1".sActBwControlIn.sInterface.SequenceRun AND #sActBwControlIn.sInterface.StartRequest AND #sShuttlePosExt),
                        iJobReq := #sActBwControlIn.sInterface.StartRequest,
                        iShuttleModeAutoPos := #tAxis_U_Position.BwLoad,
                        iShuttleModeAutoPosSetPoint := "DB_AxisPosMachinePLC".Axis_U2.BwLoad,
                        iShuttleModeSemiAutoPos := #tAxis_U_Position.BwLoad,
                        iShuttleModeSemiAutoPosSetPoint := "DB_AxisPosMachinePLC".Axis_U2.BwLoad,
                        iShuttleMoving := #iShuttleMoving,
                        iShuttleInPos := #iShuttleInPos,
                        iModeAutoPosCondition := #sActBwControlIn.iModeAutoPosCondition,
                        iModeSemiAutoPosCondition := #sActBwControlIn.iModeSemiAutoPosCondition,
                        iNoStopCondition := #sActBwControlIn.iNoStopCondition,
                        iOperatorCycleRestart := "LBP_Chan1".E_ProgRunning,
                        iNC_Stopped :=  (NOT "LBP_Chan1".E_ProgRunning AND "DB_OPC_Machine".Parameters.ConsecutiveBwIn = 0) OR "DB_OPC_Machine".Parameters.ConsecutiveBwIn > 0,
                        iNC_Running := "LBP_Chan1".E_ProgRunning,
                        iMissingPart:=#sBwControlIn.sMissingBwCtrl,
                        iExtraPart:=#sBwControlIn.sExtraBwCtrl,
                        iPLC_DateAndTime := "DB_ReadDateAndTime".sDateAndTime,
                        iStepPause := #sActBwControlIn.iStepPause, 
                        oShuttleStartReq => #sActBwControlIn.oShuttleStartReq,
                        oShuttlePosSetPoint => #sActBwControlIn.oShuttlePosSetPoint,
                        oStopNC_Req => #sActBwControlIn.oStopNC_Req,       // Implicite par Alarm Message
                        oRestartNC_Req => #sActBwControlIn.oRestartNC_Req, // Implicite par Restart NC
                        oRestartStep => #sActBwControlIn.oRestartStep,
                        oContinuationStep => #sActBwControlIn.oContinuationStep,
                        oMsgMissingPart=>#sActBwControlIn.oMsgMissingPart,
                        oMsgExtraPart=>#sActBwControlIn.oMsgExtraPart);

       IF "DB_OPC_Machine".Parameters.ConsecutiveBwIn = 0 THEN
           #sRT_BwControlInMissing(CLK := #sActBwControlIn.oMsgMissingPart);
           IF #sRT_BwControlInMissing.Q THEN
               "LBP_AlarmMsgs".UserA[03].A70UUxx[25] := TRUE;
           END_IF;

           #sRT_BwControlInExtra(CLK := #sActBwControlIn.iExtraPart);
           IF #sRT_BwControlInExtra.Q THEN
               "LBP_AlarmMsgs".UserA[03].A70UUxx[26] := TRUE;
           END_IF;
       ELSE
           "LBP_AlarmMsgs".UserA[03].A70UUxx[25] := FALSE;
           "LBP_AlarmMsgs".UserA[03].A70UUxx[26] := FALSE;
       END_IF;
   END_REGION

   REGION Axis U-V-W Start Request
       // Axis U - Start Request
       #oShuttleStartReq :=
       #sShuttleInt.oShuttleStartReq
       OR #sShuttleExt.oShuttleStartReq
       OR #sControlIn.oShuttleStartReq
       OR #sControlOut.oShuttleStartReq
       OR #sBlowing.oShuttleStartReq
       OR #sIntLoadUnload.oShuttleStartReq
       OR #sIntLoadUnloadOP.oShuttleStartReq
       OR #sExtLoadUnload.oShuttleStartReq
       OR #sBwLoadUnload.oShuttleStartReq
       OR #sBwControlIn.oShuttleStartReq
       OR #sActPartControlIn.oShuttleStartReq
       OR #sActPartControlout.oShuttleStartReq
       OR #sActBwControlIn.oShuttleStartReq;

       // Axis U - Position Set point according to start request
       IF #sShuttleInt.oShuttleStartReq THEN
           #oShuttlePosSetPoint := #sShuttleInt.oShuttlePosSetPoint;
       ELSIF #sShuttleExt.oShuttleStartReq THEN
           #oShuttlePosSetPoint := #sShuttleExt.oShuttlePosSetPoint;
       ELSIF #sControlIn.oShuttleStartReq THEN
           #oShuttlePosSetPoint := #sControlIn.oShuttlePosSetPoint;
       ELSIF #sControlOut.oShuttleStartReq THEN
           #oShuttlePosSetPoint := #sControlOut.oShuttlePosSetPoint;
       ELSIF #sExtLoadUnload.oShuttleStartReq THEN
           #oShuttlePosSetPoint := #sExtLoadUnload.oShuttlePosSetPoint;
       ELSIF #sIntLoadUnload.oShuttleStartReq THEN
           #oShuttlePosSetPoint := #sIntLoadUnload.oShuttlePosSetPoint;
       ELSIF #sIntLoadUnloadOP.oShuttleStartReq THEN
           #oShuttlePosSetPoint := #sIntLoadUnloadOP.oShuttlePosSetPoint;
       ELSIF #sBwLoadUnload.oShuttleStartReq THEN
           #oShuttlePosSetPoint := #sBwLoadUnload.oShuttlePosSetPoint;
       ELSIF #sBwControlIn.oShuttleStartReq THEN
           #oShuttlePosSetPoint := #sBwControlIn.oShuttlePosSetPoint;
       ELSIF #sActPartControlIn.oShuttleStartReq THEN
           #oShuttlePosSetPoint := #sActPartControlIn.oShuttlePosSetPoint;
       ELSIF #sActPartControlout.oShuttleStartReq THEN
           #oShuttlePosSetPoint := #sActPartControlout.oShuttlePosSetPoint;
       ELSIF #sActBwControlIn.oShuttleStartReq THEN
           #oShuttlePosSetPoint := #sActBwControlIn.oShuttlePosSetPoint;
       ELSIF  #sBlowing.oShuttleStartReq THEN
           #oShuttlePosSetPoint := #sBlowing.oShuttlePosSetPoint;
       ELSE
           #oShuttleStartReq := FALSE;
       END_IF;

       // Axis V - Start Request
       #oAxisVStartReq :=
       #sIntLoadUnload.oAxisV_StartReq
       OR #sIntLoadUnloadOP.oAxisV_StartReq
       OR #sBlowing.oAxisV_StartReq;

       // Axis V - Position Set point  according to start request
       IF #sIntLoadUnload.oAxisV_StartReq THEN
           #oAxisVPosSetPoint := #sIntLoadUnload.oAxisV_PosSetPoint;
       ELSIF #sIntLoadUnloadOP.oAxisV_StartReq THEN
           #oAxisVPosSetPoint := #sIntLoadUnloadOP.oAxisV_PosSetPoint;
       ELSIF #sBlowing.oAxisV_StartReq THEN
           #oAxisVPosSetPoint := #sBlowing.oAxisV_PosSetPoint;
       ELSE
           #oAxisVStartReq := FALSE;
       END_IF;

       // Axis W - Start Request
       #oAxisWStartReq :=
       #sIntLoadUnload.oAxisW_StartReq
       OR #sIntLoadUnloadOP.oAxisW_StartReq
       OR #sBlowing.oAxisW_StartReq;

       // Axis W - Position Set point  according to start request
       IF #sIntLoadUnload.oAxisW_StartReq THEN
           #oAxisWPosSetPoint := #sIntLoadUnload.oAxisW_PosSetPoint;
       ELSIF #sIntLoadUnloadOP.oAxisW_StartReq THEN
           #oAxisWPosSetPoint := #sIntLoadUnloadOP.oAxisW_PosSetPoint;
       ELSIF #sBlowing.oAxisW_StartReq THEN
           #oAxisWPosSetPoint := #sBlowing.oAxisW_PosSetPoint;
       ELSE
           #oAxisWStartReq := FALSE;
       END_IF;
   END_REGION

   REGION Gates Command Request
       // External Gate
       #oExtGateOpenReq := #sShuttleInt.oExtGateOpenReq OR #sShuttleExt.oExtGateOpenReq;
       #oExtGateCloseReq := #sShuttleInt.oExtGateCloseReq OR #sShuttleExt.oExtGateCloseReq;

       // Internal Gate
       #oIntGateOpenReq := #sShuttleInt.oIntGateOpenReq OR #sShuttleExt.oIntGateOpenReq;
       #oIntGateCloseReq := #sShuttleInt.oIntGateCloseReq OR #sShuttleExt.oIntGateCloseReq;
   END_REGION

   REGION Gripper Command Request
       // Load Gripper
       #oLoadGripperCloseReq := #sIntLoadUnload.oLoadGripperCloseReq
       OR #sIntLoadUnloadOP.oLoadGripperCloseReq;
       // Unload Gripper
       #oUnloadGripperOpenReq := #sIntLoadUnload.oUnloadGripperOpenReq
       OR #sIntLoadUnloadOP.oUnloadGripperOpenReq;
   END_REGION

   REGION Blowing Command Request
       #oBlowingReq := #sBlowing.oBlowingReq;
   END_REGION
END_FUNCTION_BLOCK
